(* PLC project , Danfoss PLUS+1 GUIDE 2025.3.3.6907 *)
(* stored: creationDateTime 2026-05-25T10:52:25, modificationDateTime 2026-05-25T11:42:11 *)

FUNCTION_BLOCK FB_encriptTSM_Tool
  VAR_INPUT
    acc_x : INT;
    acc_y : INT;
    acc_z : INT;
  END_VAR
  VAR_OUTPUT
    pitch : REAL;
    roll : REAL;
    pitchInt : INT;
    rollInt : INT;
  END_VAR
  VAR
    norm : REAL;
    ax_norm : REAL;
    ay_norm : REAL;
    az_norm : REAL;
    x_r : REAL;
    y_r : REAL;
    z_r : REAL;
  END_VAR

            


x_r := INT_TO_REAL(acc_x);
y_r := INT_TO_REAL(acc_y);
z_r := INT_TO_REAL(acc_z);

norm := SQRT(
    x_r * x_r +
    y_r * y_r +
    z_r * z_r
);

IF norm > 0.0 THEN

    ax_norm := y_r / norm;
    ay_norm := x_r / norm;
    az_norm := z_r / norm;

    roll := ATAN2(
        ax_norm,
        SQRT(ay_norm * ay_norm + az_norm * az_norm)
    ) * 180.0 / 3.141592653589793;

    pitch := ATAN2(
        ay_norm,
        SQRT(ax_norm * ax_norm + az_norm * az_norm)
    ) * 180.0 / 3.141592653589793;
    
    rollInt:= REAL_TO_INT(roll*100)*-1;
    pitchInt:=REAL_TO_INT(pitch*100)*-1;

ELSE

    pitch := 0.0;
    roll  := 0.0;
    
    pitchInt:=0;
    rollInt:=0;

END_IF;
          
END_FUNCTION_BLOCK
